FUNCTION_BLOCK ABSTRACT ZAppSequence EXTENDS ZApplication.Sequence IMPLEMENTS ZCore.ISequence

METHOD StepDecoded : ZCore.ZString
VAR_INPUT
  stepIndex : INT;
END_VAR
VAR_INST
  _stepIndexDecoded : ZAppStep;
END_VAR
_stepIndexDecoded := stepIndex;
StepDecoded := TO_STRING(_stepIndexDecoded);
END_METHOD

END_FUNCTION_BLOCK

(* stored: Version 1.1.0.1
   POU ZAppSequence: Id {5bf84154-0fcb-41b0-a47c-81d4ed4d16c9}, SpecialFunc None
   Method StepDecoded: Id {841d67e8-d280-4eec-a0a9-6d4d12816c69} *)
